// TIA Portal V17 export
// export: Created 2025-06-25T13:13:29.5089042Z, ExportSetting WithDefaults, DisplayName Totally Integrated Automation Portal, DisplayVersion V17 Update 8, DisplayName TIA Portal Openness, DisplayVersion V17 Update 8, DisplayName TIA Portal Version Control Interface, DisplayVersion V17, DisplayName STEP 7 Professional, DisplayVersion V17 Update 8, DisplayName STEP 7 Safety, DisplayVersion V17 Update 6, DisplayName WinCC Advanced, DisplayVersion V17 Update 8
TYPE "stHoursCounter"
// stored: IsFailsafeCompliant false
   STRUCT
      nHours : UDInt;   // 0-4294967295
      nMinutes : USInt;   // 0-59
      nSeconds : USInt;   // 0-59
      bReset : Bool;   // Command bit to reset the count
   END_STRUCT;
END_TYPE
